(* CoDeSys 2.3.9.41 project: Teplo.pro *)
(* Libraries: STANDARD.LIB 4.10.05 10:14:46, IECSFC.LIB 13.4.06 14:51:28, SYSLIBTIME.LIB 20.2.06 12:31:16, SYSTASKINFO.LIB 20.2.06 12:31:38, ANALYZATION.LIB 5.10.99 08:05:06, SYSLIBCALLBACK.LIB 20.2.06 12:31:08 *)

(* PLC configuration (modules and I/O channels)
Fast discrete inputs [I_SIMPLE_INPUT] node 0, in %IB0 out %QB0 {Filtrationtime = 10}
  AT %IX0.0 [BitInput] Discrete input 1
  AT %IX0.1 [BitInput] Discrete input 2
  AT %IX0.2 [BitInput] Discrete input 3
  AT %IX0.3 [BitInput] Discrete input 4
Discrete inputs [ID130] node 1, in %IB1 out %QB1 {Filtrationtime_GeneralINP = 10; Visibility = No; PinCount = 12}
  AT %IB1.0 [ByteInput] 8 discrete inputs
  AT %IB1.1 [ByteInput] 4 discrete inputs
Discrete outputs [ID131] node 2, in %IB2 out %QB2 {SafeValueByte = 0; SafeValueByteM = 0; Visibility = No; PinCount = 12}
  AT %QB2.0 [ByteOutput] 8 discrete outputs
  AT %QB2.1 [ByteOutput] 4 discrete outputs
Fast analog inputs [ID125] node 3, in %IB3 out %QB3 {Flt_Comm = 50Hz 2Por}
  AT %IR3.0 [FloatInputP] AI #1 {AIN_TYPE = 4-20 mA; Peak_Filtr = 200; Flt_Ch = Off; TauRC = 10; MinFV = 0; MaxFV = 20000.0}
  AT %IR3.1 [FloatInputP] AI #2 {AIN_TYPE = 4-20 mA; Peak_Filtr = 200; Flt_Ch = Off; TauRC = 10; MinFV = 0; MaxFV = 20000.0}
  AT %IR3.2 [FloatInputP] AI #3 {AIN_TYPE = 4-20 mA; Peak_Filtr = 200; Flt_Ch = Off; TauRC = 10; MinFV = 0; MaxFV = 20000.0}
  AT %IR3.3 [FloatInputP] AI #4 {AIN_TYPE = 4-20 mA; Peak_Filtr = 200; Flt_Ch = Off; TauRC = 10; MinFV = 0; MaxFV = 20000.0}
  AT %IR3.4 [FloatInputP] AI #5 {AIN_TYPE = 4-20 mA; Peak_Filtr = 200; Flt_Ch = Off; TauRC = 10; MinFV = 0; MaxFV = 20000.0}
  AT %IR3.5 [FloatInputP] AI #6 {AIN_TYPE = 4-20 mA; Peak_Filtr = 200; Flt_Ch = Off; TauRC = 10; MinFV = 0; MaxFV = 20000.0}
  AT %IR3.6 [FloatInputP] AI #7 {AIN_TYPE = 4-20 mA; Peak_Filtr = 200; Flt_Ch = Off; TauRC = 10; MinFV = 0; MaxFV = 20000.0}
  AT %IR3.7 [FloatInputP] AI #8 {AIN_TYPE = 4-20 mA; Peak_Filtr = 200; Flt_Ch = Off; TauRC = 10; MinFV = 0; MaxFV = 20000.0}
  AT %IW3.8 [WordInput] AI read time (10ms)
Analog outputs [ID126] node 4, in %IB4 out %QB4
  AT %QR4.0 [FloatOutputP] AO #1 {AOUT_TYPE = 4-20 mA; SafeValueREAL = 0.0}
  AT %QR4.1 [FloatOutputP] AO #2 {AOUT_TYPE = 4-20 mA; SafeValueREAL = 0.0}
  AT %QR4.2 [FloatOutputP] AO #3 {AOUT_TYPE = 4-20 mA; SafeValueREAL = 0.0}
  AT %QR4.3 [FloatOutputP] AO #4 {AOUT_TYPE = 4-20 mA; SafeValueREAL = 0.0}
Special input [ID103] node 5, in %IB5 out %QB5 {Filtrationtime = 1000; PinCount = 1; WatchDogPeriod = 400; PollPeriod = 3000; Visibility = No}
  AT %IX5.0 [BitInput] Special input
Special output [ID104] node 6, in %IB6 out %QB6 {Visibility = No; PinCount = 1}
  AT %QX6.0 [BitOutput] Special output
AT %QD7.0 [DWordOutput] Last address
AT %QW7.1 [WordOutput] Last error
RS-485-1 [COM1_USART] node 0, in %IB7.0 out %QB7.0 {CommunicationSpeed = 11520; Parity = NO PARITY CHECK; BitLength = 8 bits; StopLength = Two stop bits; InterfaceType = RS485; FrameOriented = RTU; Timeout = 0; Visibility = No}
AT %QB7.1.0 [ComChannel] Command (0xff - Start)
AT %IW7.1.0.0 [WordInput] уставка 1
AT %IW7.1.1.0 [WordInput] температура 1
AT %QW7.1.2.0 [WordOutput] запись уставки 1
AT %IW7.1.3.0 [WordInput] состояние 1
Universal Modbus device [ID2000] node 2, in %IB7.2 out %QB7.2 {ModuleIP = 10:0:0:223; ServiceTimeout = 150; TCPport = 502; NetMode = Serial; ModuleSlaveAddress = 4; RequestType = By poll time; PeriodOfService = 3000; Visibility = No; RepeatCounter = 0; ByteSequence = Native}
  AT %QB7.2.0 [ComChannel] Command (0xff - Start)
AT %IW7.2.0.0 [WordInput] уставка 2
AT %IW7.2.1.0 [WordInput] температура 2
AT %QW7.2.2.0 [WordOutput] запись уставки 2
AT %IW7.2.3.0 [WordInput] состояние 2
AT %QB7.3.0 [ComChannel] Command (0xff - Start)
AT %ID7.3.0.0 [DWordInput] уст. (рег для записи 20209)
AT %ID7.3.1.0 [DWordInput] мощность 00.00
AT %IW7.3.2.0 [WordInput] напряжение 000.0
AT %IW7.3.3.0 [WordInput] частота 00.0
AT %ID7.3.4.0 [DWordInput] ток 00.00
AT %ID7.3.5.0 [DWordInput] давление 0.000
AT %QD7.3.6.0 [DWordOutput] задание уставки
RS-232 [COM2_USART] node 0, in %IB8.0.0 out %QB8.0.0 {CommunicationSpeed = 11520; Parity = EVEN; BitLength = 8 bits; StopLength = One stop bit; InterfaceType = RS232; FrameOriented = RTU; Timeout = 0; Visibility = No}
8 bits [8Bit] node 1, in %IB8.1 out %QB8.1
  AT %QB8.1.0 [ByteOutput]
2 byte [Register] node 2, in %IB8.2 out %QB8.2
  AT %QW8.2.0 [WordOutput] температура 1
2 byte [Register] node 3, in %IB8.3 out %QB8.3
  AT %QW8.3.0 [WordOutput] уставка 1
2 byte [Register] node 4, in %IB8.4 out %QB8.4
  AT %QW8.4.0 [WordOutput] температура 2
  AT %QW8.5.0 [WordOutput] уставка 2
AT %QD8.6.0 [DWordOutput] уставка пч
AT %QD8.7.0 [DWordOutput] мощность
AT %QW8.8.0 [WordOutput] напряжение
AT %QW8.9.0 [WordOutput] частота
AT %QD8.10.0 [DWordOutput] ток
AT %QD8.11.0 [DWordOutput] давление
AT %QW9.0 [W32WordOutput] Status
AT %QW9.0.0 [WordOutput]
AT %QW9.1.0 [WordOutput] t1
AT %QW9.2.0 [WordOutput] t2
AT %QD9.3.0 [DWordOutput] P
Modbus [MODBUS_ID302] node 0, in %IB10.0 out %QB10.0
  TCP [TCP_ID221] node 0, in %IB10.0.0 out %QB10.0.0 {RemotePort = 502; Visibility = No}
2 byte [Register] node 1, in %IB10.1 out %QB10.1
  AT %QW10.1.0 [WordOutput] T1
2 byte [Register] node 2, in %IB10.2 out %QB10.2
  AT %QW10.2.0 [WordOutput] sT1
2 byte [Register] node 3, in %IB10.3 out %QB10.3
  AT %QW10.3.0 [WordOutput] S1
2 byte [Register] node 4, in %IB10.4 out %QB10.4
  AT %QW10.4.0 [WordOutput] T2
2 byte [Register] node 5, in %IB10.5 out %QB10.5
  AT %QW10.5.0 [WordOutput] sT2
2 byte [Register] node 6, in %IB10.6 out %QB10.6
  AT %QW10.6.0 [WordOutput] S2
2 byte [Register] node 7, in %IB10.7 out %QB10.7
  AT %QW10.7.0 [WordOutput] Volt
2 byte [Register] node 8, in %IB10.8 out %QB10.8
  AT %QW10.8.0 [WordOutput] Freq
4 byte [FourBytes] node 9, in %IB10.9 out %QB10.9
  AT %QD10.9.0 [DWordOutput] уставка
  AT %QD10.10.0 [DWordOutput] мощность
  AT %QD10.11.0 [DWordOutput] ток
  AT %QD10.12.0 [DWordOutput] давление
*)

(* Global variable list: Global_Variables *)
VAR_GLOBAL
(*ТРМ 1*)
	(*Состояние выхода*)
	Stat_Pan_1 AT %QX8.1.0.0 : BOOL;	(*передача на панель*)
	Stat_trm_1 AT %IW7.1.3.0 : WORD;	(*чтение с ТРМ'а*)

	(*температура и уставка*)
	T_panel1 AT %QW8.2.0 : WORD;
	T_trm1 AT %IW7.1.1.0 : WORD;
	Ts_panel1 AT %QW8.3.0 : WORD;
	Ts_trm1 AT %IW7.1.0.0 : WORD;

	(*задание уставки*)
	T_set1 AT %QW7.1.2.0 : WORD;

(*ТРМ 2*)
	(*Состояние выхода*)
	Stat_Pan_2 AT %QX8.1.0.1 : BOOL;	(*передача на панель*)
	Stat_trm_2 AT %IW7.2.3.0 : WORD;	(*чтение с ТРМ'а*)

	(*температура и уставка*)
	T_panel2 AT %QW8.4.0 : WORD;
	T_trm2 AT %IW7.2.1.0 : WORD;
	Ts_panel2 AT %QW8.5.0 : WORD;
	Ts_trm2 AT %IW7.2.0.0 : WORD;

	(*задание уставки*)
	T_set2 AT %QW7.2.2.0 : WORD;

(*задвижка*)
	Valve1 AT %QX8.1.0.2 : BOOL;
	Valve2 AT %QX8.1.0.3 : BOOL;

(*проверка связи*)
	Connection : INT;

(*пч*)
	(*для панели*)
	Ps_panel AT %QD8.6.0 : DWORD;
	Power_panel AT %QD8.7.0 : DWORD;
	Volt_panel AT %QW8.8.0 : WORD;
	Freq_panel AT %QW8.9.0 : WORD;
	Curr_panel AT %QD8.10.0 : DWORD;
	P_panel AT %QD8.11.0 : DWORD;

	(*с пч*)
	Ps_fc AT %ID7.3.0.0 : DWORD;
	Power_fc AT %ID7.3.1.0 : DWORD;
	Volt_fc AT %IW7.3.2.0 : WORD;
	Freq_fc AT %IW7.3.3.0 : WORD;
	Curr_fc AT %ID7.3.4.0 : DWORD;
	P_fc AT %ID7.3.5.0 : DWORD;

	(*на пч*)
	P_set AT %QD7.3.6.0 : DWORD;

(*архивы-архивчики*)
	T1_arch AT %QW9.1.0 : WORD;
	T2_arch AT %QW9.2.0 : WORD;
	P_arch AT %QD9.3.0 : DWORD;

(*delphi*)
	dT_trm1 AT %QW10.1.0 : WORD;
	dTs_trm1 AT %QW10.2.0 : WORD;
	dStat_trm_1 AT %QW10.3.0 : WORD;

	dT_trm2 AT %QW10.4.0 : WORD;
	dTs_trm2 AT %QW10.5.0 : WORD;
	dStat_trm_2 AT %QW10.6.0 : WORD;


	dVolt_fc AT %QW10.7.0 : WORD;
	dFreq_fc AT %QW10.8.0 : WORD;

	dPs_fc AT %QD10.9.0 : DWORD;
	dPower_fc AT %QD10.10.0 : DWORD;

	dCurr_fc AT %QD10.11.0 : DWORD;
	dP_fc AT %QD10.12.0 : DWORD;


END_VAR

(* POU PLC_PRG, ST *)
PROGRAM PLC_PRG
VAR


END_VAR
(*________ТРМ 1_________*)

(*передача ТРМ -> панель*)
T_panel1 := T_trm1;

(*изменение уставки*)
IF Ts_panel1 <> Ts_trm1
	THEN T_set1 := Ts_panel1;
END_IF;

(*состояние выхода*)
IF Stat_trm_1 = 1000
	THEN Stat_Pan_1 := 1;
		ELSE Stat_Pan_1 := 0;
END_IF;

(*_________ТРМ 2______*)

(*передача ТРМ -> панель*)
T_panel2 := T_trm2;

(*изменение уставки*)
IF Ts_panel2 <> Ts_trm2
	THEN T_set2 := Ts_panel2;
END_IF;

(*состояние выхода*)
IF Stat_trm_2 = 1000
	THEN Stat_Pan_2 := 1;
		ELSE Stat_Pan_2 := 0;
END_IF;

(*_______Задвижки______*)

IF Stat_Pan_1
	THEN Valve1 := 0;
		ELSE Valve1 := 1;
END_IF;

IF Stat_Pan_2
	THEN Valve2 := 0;
		ELSE Valve2 := 1;
END_IF;

(*_____Connection____*)
IF Connection=1
	THEN Connection := 2;
END_IF;

(*передача ПЧ -> панель*)
Power_panel := Power_fc;
Volt_panel := Volt_fc;
Freq_panel := Freq_fc;
Curr_panel := Curr_fc;
P_panel := P_fc;

(*задание уставки*)
IF Ps_panel <> Ps_fc
	THEN P_set := Ps_panel;
END_IF;


(*архивы-архивчики*)
T1_arch := T_trm1;
T2_arch := T_trm2;
P_arch :=	P_fc;


(*delphi*)
	dT_trm1 := T_trm1;
	dTs_trm1 := Ts_trm1;
	dStat_trm_1 := Stat_trm_1;

	dT_trm2 := T_trm2;
	dTs_trm2 := Ts_trm2;
	dStat_trm_2 := Stat_trm_2;


	dVolt_fc  := Volt_fc;
	dFreq_fc := Freq_fc;

	dPs_fc := Ps_fc;
	dPower_fc := Power_fc;

	dCurr_fc := Curr_fc;
	dP_fc := P_fc;
END_PROGRAM
